FUNCTION_BLOCK skGoToLeft (* Composite Function Block Type *)
  (* Standard: 61499-2 *)
  (* Version 0.0, 11/8/2025, vv263, template *)
  PACKAGE Main;
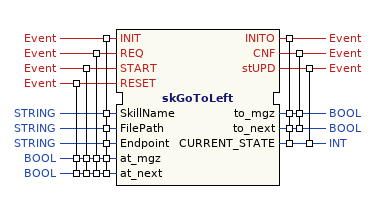
  EVENT_INPUT
    INIT WITH SkillName, FilePath, Endpoint, at_mgz, at_next; (* Initialization Request *)
    REQ WITH at_mgz, at_next; (* Normal Execution Request *)
    START WITH at_mgz, at_next;
    RESET WITH at_mgz, at_next;
  END_EVENT
  EVENT_OUTPUT
    INITO WITH to_mgz, to_next, CURRENT_STATE; (* Initialization Confirm *)
    CNF WITH to_mgz, to_next; (* Execution Confirmation *)
    stUPD WITH CURRENT_STATE;
  END_EVENT
  VAR_INPUT
    SkillName : STRING;
    FilePath : STRING;
    Endpoint : STRING;
    at_mgz : BOOL;
    at_next : BOOL;
  END_VAR
  VAR_OUTPUT
    to_mgz : BOOL;
    to_next : BOOL;
    CURRENT_STATE : INT;
  END_VAR
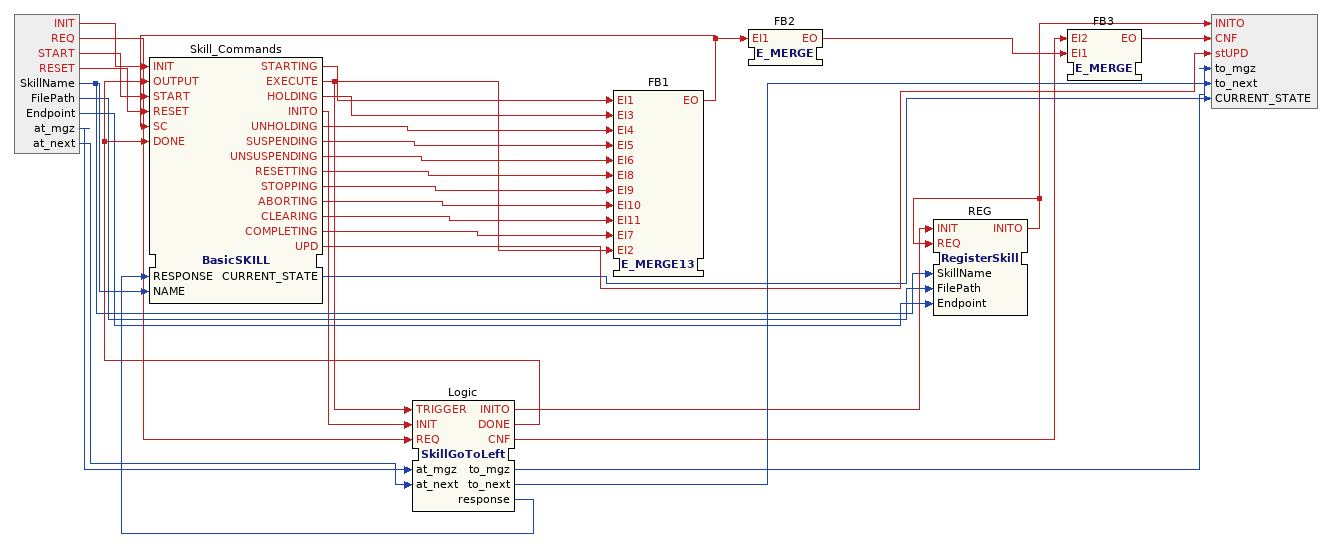
  FBS
    Skill_Commands : BasicSKILL;
    REG : RegisterSkill;
    Logic : SkillGoToLeft;
    FB1 : E_MERGE13;
    FB2 : E_MERGE;
    FB3 : E_MERGE;
  END_FBS
  EVENT_CONNECTIONS
    Skill_Commands.STARTING TO FB1.EI1;
    Skill_Commands.EXECUTE TO Logic.TRIGGER;
    Skill_Commands.HOLDING TO FB1.EI3;
    INIT TO Skill_Commands.INIT;
    Skill_Commands.INITO TO Logic.INIT;
    Logic.INITO TO REG.INIT;
    REG.INITO TO REG.REQ;
    REQ TO Logic.REQ;
    REG.INITO TO INITO;
    FB1.EO TO FB2.EI1;
    Skill_Commands.UNHOLDING TO FB1.EI4;
    Skill_Commands.SUSPENDING TO FB1.EI5;
    Skill_Commands.UNSUSPENDING TO FB1.EI6;
    Skill_Commands.RESETTING TO FB1.EI8;
    Skill_Commands.STOPPING TO FB1.EI9;
    Skill_Commands.ABORTING TO FB1.EI10;
    Skill_Commands.CLEARING TO FB1.EI11;
    Logic.DONE TO Skill_Commands.OUTPUT;
    START TO Skill_Commands.START;
    RESET TO Skill_Commands.RESET;
    Skill_Commands.COMPLETING TO FB1.EI7;
    Logic.CNF TO FB3.EI2;
    FB1.EO TO Skill_Commands.SC;
    Skill_Commands.EXECUTE TO FB1.EI2;
    FB3.EO TO CNF;
    FB2.EO TO FB3.EI1;
    Logic.DONE TO Skill_Commands.DONE;
    Skill_Commands.UPD TO stUPD;
  END_CONNECTIONS
  DATA_CONNECTIONS
    SkillName TO REG.SkillName;
    FilePath TO REG.FilePath;
    Endpoint TO REG.Endpoint;
    at_mgz TO Logic.at_mgz;
    at_next TO Logic.at_next;
    Logic.to_mgz TO to_mgz;
    Logic.to_next TO to_next;
    Logic.response TO Skill_Commands.RESPONSE;
    SkillName TO Skill_Commands.NAME;
    Skill_Commands.CURRENT_STATE TO CURRENT_STATE;
  END_CONNECTIONS
END_FUNCTION_BLOCK
